// TIA Portal V21 export
FUNCTION "Main stazioni" : Void   // FC26, LAD
{ S7_Optimized_Access := 'TRUE' }
// stored: SetENOAutomatically false
   VAR CONSTANT
      NonPresente : Int := 0;
      Disabilitata : Bool := 0;
      NessunConsenso : Bool := 1;
      NonRaggiunta : Byte := 2;
      Raggiunta : Byte := 1;
      Completa : Byte := 0;
      SoloStato : Byte := 1;
   END_VAR
BEGIN

REGION Network 1 (SCL): Gestione stazione - PompaAcidificazioneVascaEvaporati
   // //Parametrizzazione stazione
   // "Percorso".Stazione["K_Stazione_PompaAcidificazioneVascaEvaporati"].Prm.CadutaChiamata.DaAnalogicaPer.SogliaMini := #NonRaggiunta;

   // //Richiamo stazione
   // "GestStazione"(ConsensoMacchina:= #NessunConsenso,
   //                FermaChiamata := #Disabilitata,
   //                K_Stazione := "K_Stazione_PompaAcidificazioneVascaEvaporati",
   //                K_StazionePartner1:=#NonPresente,
   //                K_StazionePartner2:=#NonPresente,
   //                K_Analogica := "K_Analogica_LivelloSerbatoioAcidoCitrico",
   //                K_Paratia := #NonPresente,
   //                K_Motore1 := #NonPresente,
   //                K_Motore2 := "K_Pompa_Citrico_Vasca_Evaporati");

   // //Definizione dei percorsi possibili per la stazione
   // "Percorso".Stazione["K_Stazione_PompaAcidificazioneVascaEvaporati"].Destinazione["K_Stazione_VascaEvaporati"].IN.Possibile := True;

   // //Visualizzazione hmi a pannello delle strade
   // "Percorso".Hmi.Visibilità.PompaAcidificazioneVascaEvaporati.VascaEvaporati := "Percorso".Stazione["K_Stazione_PompaAcidificazioneVascaEvaporati"].Destinazione["K_Stazione_VascaEvaporati"].IN.Possibile;
END_REGION
END_FUNCTION
